TYPE AirMode : 
(
	HOLD := 0,
	IN,
	OUT,
	
	size
);
END_TYPE

(* stored: Version 1.1.0.1, ProductVersion 3.1.4024.11
   DUT AirMode: Id {173f6303-00c3-42c1-ae55-69eeefbd9f2b} *)
